FUNCTION_BLOCK StubTask IMPLEMENTS I_Task
VAR
END_VAR

{warning 'Add method implementation '}
METHOD Abort : BOOL
END_METHOD

{warning 'Add property implementation'}
PROPERTY Busy : BOOL
GET
END_GET
END_PROPERTY

{warning 'Add property implementation'}
PROPERTY Done : BOOL
GET
END_GET
END_PROPERTY

{warning 'Add property implementation'}
PROPERTY Error : BOOL
GET
END_GET
END_PROPERTY

END_FUNCTION_BLOCK

(* stored: Version 1.1.0.1
   POU StubTask: Id {c4b913a6-ffc3-4925-be97-7fe940dfab3e}, SpecialFunc None
   Method Abort: Id {43d6722c-87e6-488f-a2d8-23a304e3ae10}
   Property Busy: Id {148822db-b76d-49e4-ac90-653df4a62c57}
   Get Get: Id {9c35da09-c523-4220-b08b-ab59892c326e}
   Property Done: Id {6d0d6f9b-aebb-4d0d-8062-3bba4dc48f43}
   Get Get: Id {e33161b1-7930-4523-a05a-40c9b3664392}
   Property Error: Id {ddc0f6db-994c-4c20-ad8c-1e1474a670ba}
   Get Get: Id {88c2e8ee-f421-41cf-b239-0c98fea27289} *)
